SUBAPPLICATION DDS_SUB (* Wrapper for DDS Publisher and Subscriber Pair as a Client *)
  (* Standard: 61499-2 *)
  (* Version 1.0, 2023-03-15, Tim Hesse *)
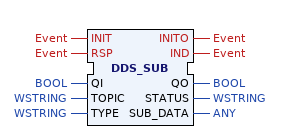
  EVENT_INPUT
    INIT; (* Initialization Request *)
    RSP; (* Application Response to IND *)
  END_EVENT
  EVENT_OUTPUT
    INITO; (* Initialization Confirm *)
    IND; (* Confirmation of Requested Service *)
  END_EVENT
  VAR_INPUT
    QI : BOOL; (* Input event qualifier *)
    TOPIC : WSTRING; (* DDS Topic *)
    TYPE : WSTRING; (* DDS Type *)
  END_VAR
  VAR_OUTPUT
    QO : BOOL; (* Output event qualifier *)
    STATUS : WSTRING; (* Service Status *)
    SUB_DATA : ANY; (* Subscribed Data *)
  END_VAR
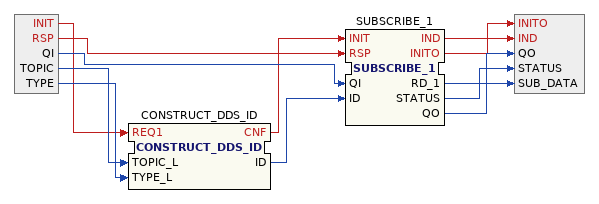
  FBS
    CONSTRUCT_DDS_ID : CONSTRUCT_DDS_ID;
    SUBSCRIBE_1 : SUBSCRIBE_1;
  END_FBS
  EVENT_CONNECTIONS
    INIT TO CONSTRUCT_DDS_ID.REQ1;
    CONSTRUCT_DDS_ID.CNF TO SUBSCRIBE_1.INIT;
    RSP TO SUBSCRIBE_1.RSP;
    SUBSCRIBE_1.IND TO IND;
    SUBSCRIBE_1.INITO TO INITO;
  END_CONNECTIONS
  DATA_CONNECTIONS
    TOPIC TO CONSTRUCT_DDS_ID.TOPIC_L;
    TYPE TO CONSTRUCT_DDS_ID.TYPE_L;
    QI TO SUBSCRIBE_1.QI;
    CONSTRUCT_DDS_ID.ID TO SUBSCRIBE_1.ID;
    SUBSCRIBE_1.RD_1 TO SUB_DATA;
    SUBSCRIBE_1.STATUS TO STATUS;
    SUBSCRIBE_1.QO TO QO;
  END_CONNECTIONS
END_SUBAPPLICATION
